// TIA Portal V20 export
DATA_BLOCK "DriveDiagInterfaceHmi"   // DB46
TITLE = DriveDiagInterfaceHmi
AUTHOR : Siemens Digital Industries
FAMILY : LAF
NAME : LAF_DriveDiagInterfaceHmi
VERSION : 1.1
// HMI interface for drive diagnostic
// stored: MemoryReserve 100
   VAR
      diagStatus : "LAF_typeDriveDiagInterfaceHmi";
      torqueLoad : Array[0.."LAF_DRV_DIAG_NO_DO"] of "LER_typeServoTorqueCalInterface";
   END_VAR
BEGIN
END_DATA_BLOCK
